TYPE ST_BufferMetadata :
	STRUCT
		headIndex	 : DINT;
		tailIndex	 : DINT;
		capacity	 : DINT;
		elementCount : DINT;
	END_STRUCT
END_TYPE

(* stored: Version 1.1.0.1, ProductVersion 3.1.4026.18
   DUT ST_BufferMetadata: Id {58158193-4b2c-454c-9283-4d2dced5c856} *)
